PROGRAM prgPD
VAR
	fbPers						: FB_WritePersistentData_General;
END_VAR

fbPers(
	eSaveModeData:= eUSVSaveMode.eSaveEventBased, 
	bLoadPersistentDataOk=> , 
	bError=> , 
	bySaveProcess=> , 
	dwStorageLast24h=> , 
	udiErrorCode=> );

END_PROGRAM

(* stored: Version 1.1.0.1, ProductVersion 3.1.4024.11
   POU prgPD: Id {8370b593-b9d2-4c0b-8b25-a99511c8c6db}, SpecialFunc None *)
